// TIA Portal V16 export
VAR_GLOBAL   // PLC tag table "Pump_IO_LAD"
   Pump_AutoMode AT %I0.0 : Bool;
   Pump_StartButton AT %I0.1 : Bool;
   Pump_StopOK AT %I0.2 : Bool;
   Pump_SafetyOK AT %I0.3 : Bool;
   Pump_OverloadOK AT %I0.4 : Bool;
   Pump_SourceWaterOK AT %I0.5 : Bool;
   Pump_LowWet AT %I0.6 : Bool;
   Pump_HighWet AT %I0.7 : Bool;
   Pump_ResetButton AT %I1.0 : Bool;
   Pump_MotorFeedback AT %I1.1 : Bool;
   Pump_PumpCmd AT %Q0.0 : Bool;
   Pump_Alarm AT %Q0.1 : Bool;
   Pump_Enabled AT %Q0.2 : Bool;
END_VAR
